// TIA Portal V15.1 export
// export: Created 2020-06-12T07:35:47.8505859Z, ExportSetting None, DisplayName Totally Integrated Automation Portal, DisplayVersion V15.1, DisplayName TIA Portal Openness, DisplayVersion V15.1, DisplayName STEP 7 Professional, DisplayVersion V15.1, DisplayName STEP 7 Safety, DisplayVersion V15.1, DisplayName WinCC Advanced, DisplayVersion V15.1
FUNCTION "DED_Line" : Void   // FC551, FBD
TITLE = Dedusting Pressure control
{ S7_Optimized_Access := 'FALSE' }
// stored: AutoNumber false, SetENOAutomatically False
   VAR_TEMP
      _csf : Bool;
      _hi : Bool;
      _bet : Bool;
      _lo : Bool;
      _cv01_init : Real;
      tVentDemand : Bool;
      _lockw : Word;
      tOpen : Bool;
      tUseIndirect : Bool;
      tLimPressure : Real;
      tCV01set : Real;
      tVarR1 : Real;
      tEnableIndirect : Bool;
      tHoodPressSet : Real;
      tContLock : Bool;
      tContAckn : Bool;
      tContIsOn : Bool;
      tContIsLocked : Bool;
      tContHasFault : Bool;
      tPressAboveSet : Real;
      tDPhigh : Real;
      tCV01set2 : Real;
   END_VAR
   VAR_TEMP   // added for the SCL form of the ladder/FBD networks
      _w1 : Bool;
   END_VAR
BEGIN

REGION Network 1: COMMON SYSTEM FAULT
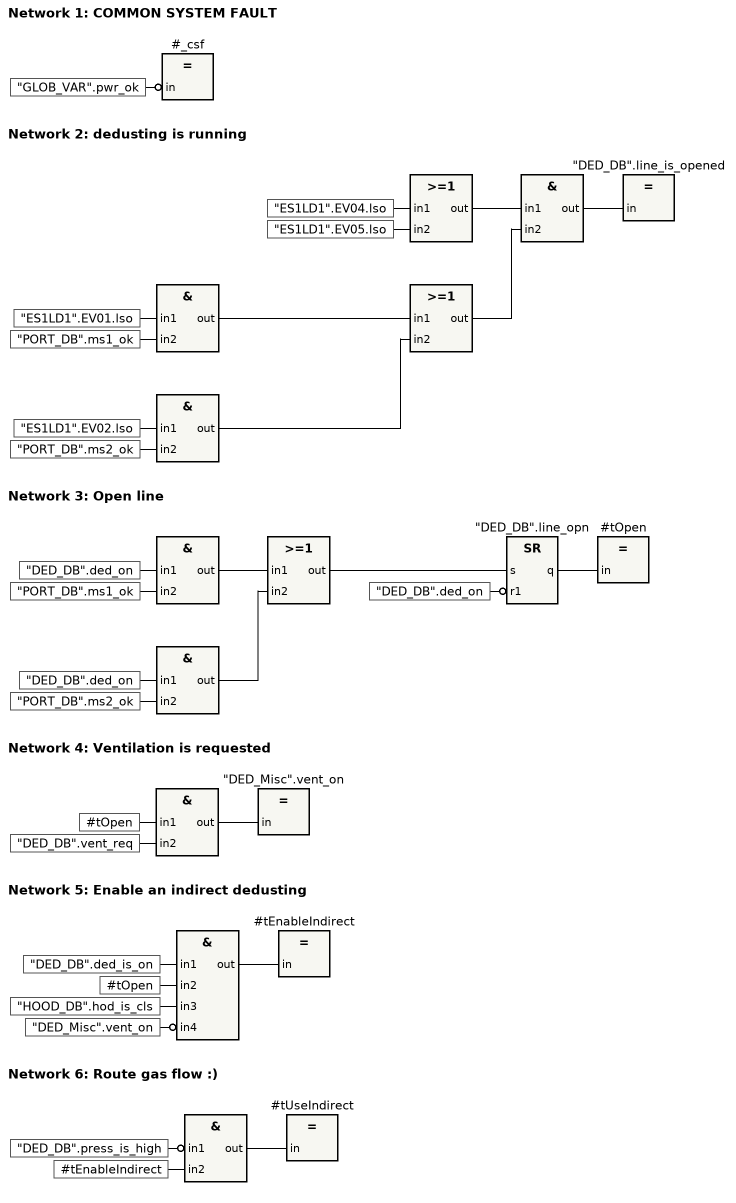
   #_csf := NOT "GLOB_VAR".pwr_ok;
END_REGION

REGION Network 2: dedusting is running
   "DED_DB".line_is_opened := ("ES1LD1".EV04.lso OR "ES1LD1".EV05.lso) AND (("ES1LD1".EV01.lso AND "PORT_DB".ms1_ok) OR ("ES1LD1".EV02.lso AND "PORT_DB".ms2_ok));
END_REGION

REGION Network 3: Open line
   IF ("DED_DB".ded_on AND "PORT_DB".ms1_ok) OR ("DED_DB".ded_on AND "PORT_DB".ms2_ok) THEN
       "DED_DB".line_opn := TRUE;   // SR flip-flop
   END_IF;
   IF NOT "DED_DB".ded_on THEN "DED_DB".line_opn := FALSE; END_IF;
   #tOpen := "DED_DB".line_opn;
END_REGION

REGION Network 4: Ventilation is requested
   "DED_Misc".vent_on := #tOpen AND "DED_DB".vent_req;
END_REGION

REGION Network 5: Enable an indirect dedusting
   #tEnableIndirect := "DED_DB".ded_is_on AND #tOpen AND "HOOD_DB".hod_is_cls AND NOT "DED_Misc".vent_on;
END_REGION

REGION Network 6: Route gas flow :)
   #tUseIndirect := NOT "DED_DB".press_is_high AND #tEnableIndirect;
END_REGION

REGION Network 7: Pressure Tresholds calculation
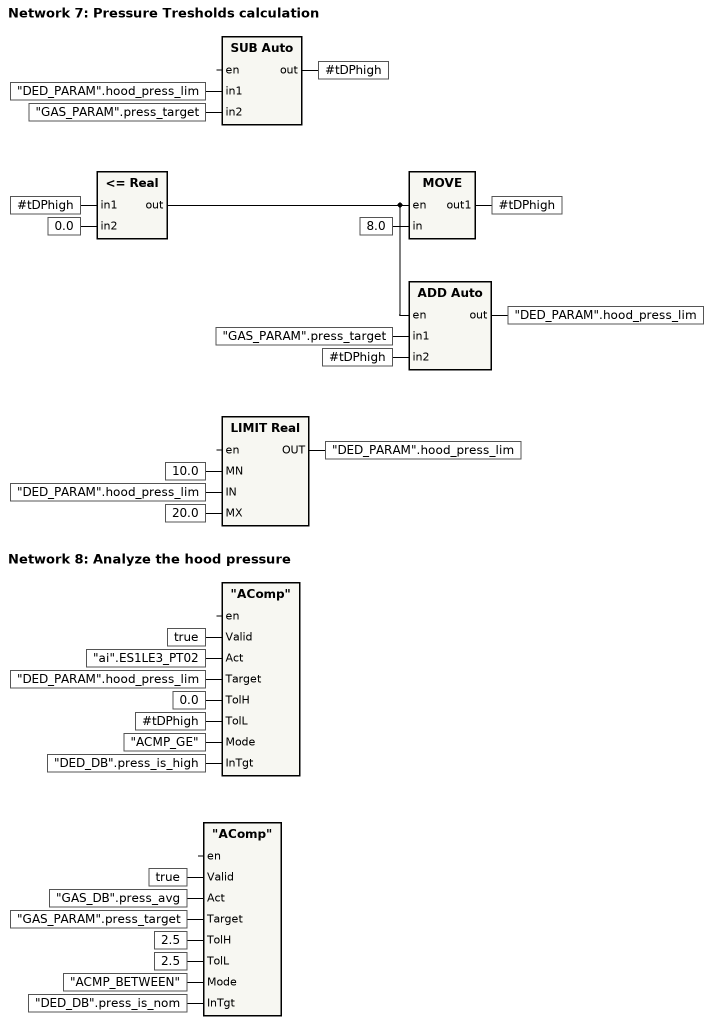
   #tDPhigh := "DED_PARAM".hood_press_lim - "GAS_PARAM".press_target;
   #_w1 := #tDPhigh <= 0.0;
   IF #_w1 THEN
       #tDPhigh := 8.0;
       "DED_PARAM".hood_press_lim := "GAS_PARAM".press_target + #tDPhigh;
   END_IF;
   "DED_PARAM".hood_press_lim := LIMIT(MN := 10.0, IN := "DED_PARAM".hood_press_lim, MX := 20.0);
END_REGION

REGION Network 8: Analyze the hood pressure
   "AComp"(Valid := true,
           Act := "ai".ES1LE3_PT02,
           Target := "DED_PARAM".hood_press_lim,
           TolH := 0.0,
           TolL := #tDPhigh,
           Mode := "ACMP_GE",
           InTgt := "DED_DB".press_is_high);
   "AComp"(Valid := true,
           Act := "GAS_DB".press_avg,
           Target := "GAS_PARAM".press_target,
           TolH := 2.5,
           TolL := 2.5,
           Mode := "ACMP_BETWEEN",
           InTgt := "DED_DB".press_is_nom);
END_REGION

REGION Network 9: Detect the pressure
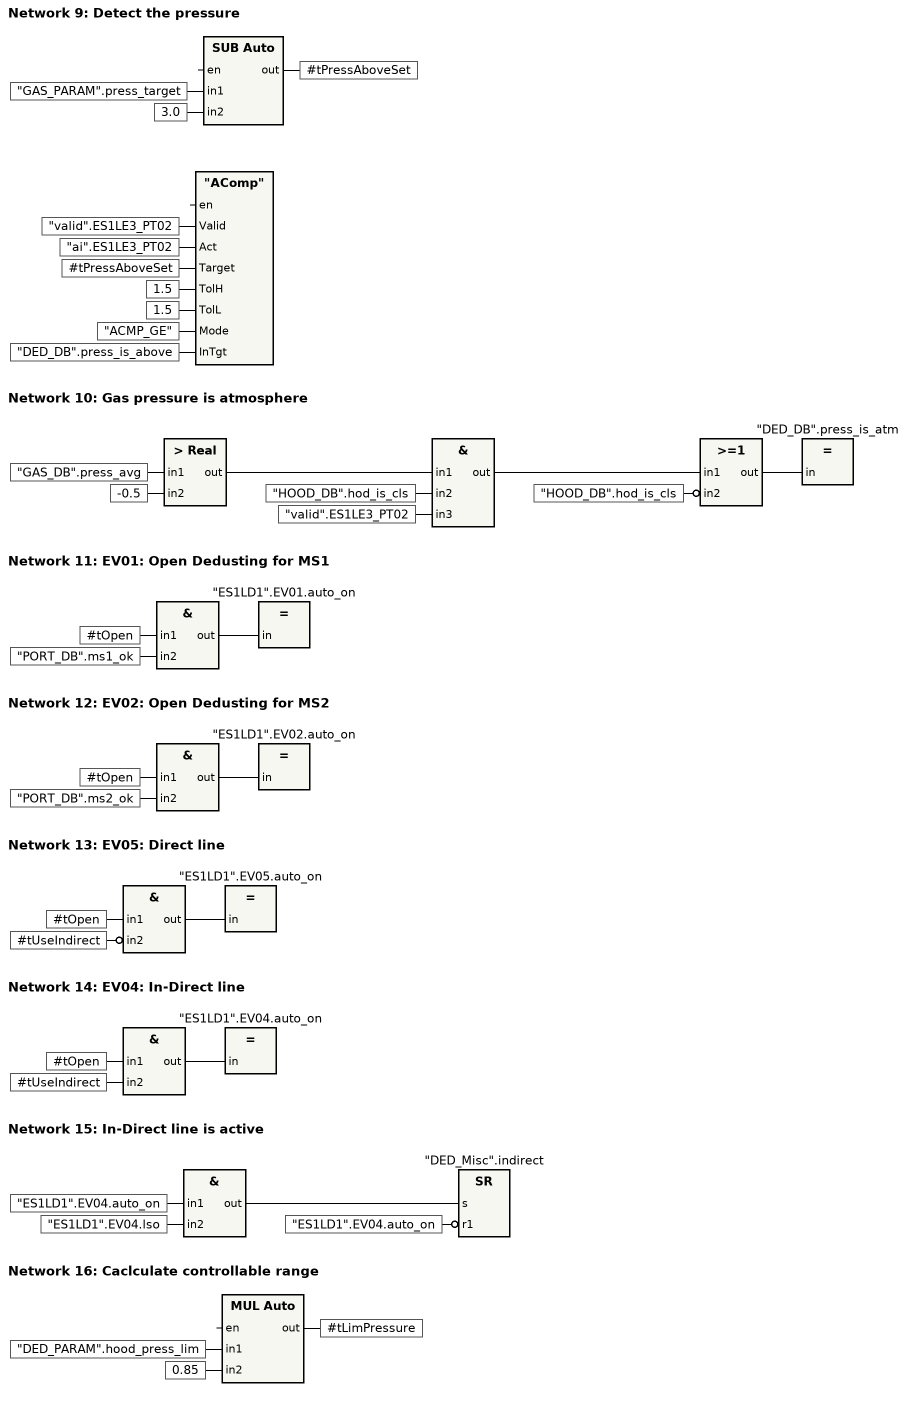
   #tPressAboveSet := "GAS_PARAM".press_target - 3.0;
   "AComp"(Valid := "valid".ES1LE3_PT02,
           Act := "ai".ES1LE3_PT02,
           Target := #tPressAboveSet,
           TolH := 1.5,
           TolL := 1.5,
           Mode := "ACMP_GE",
           InTgt := "DED_DB".press_is_above);
END_REGION

REGION Network 10: Gas pressure is atmosphere
   "DED_DB".press_is_atm := (("GAS_DB".press_avg > (-0.5)) AND "HOOD_DB".hod_is_cls AND "valid".ES1LE3_PT02) OR NOT "HOOD_DB".hod_is_cls;
END_REGION

REGION Network 11: EV01: Open Dedusting for MS1
   "ES1LD1".EV01.auto_on := #tOpen AND "PORT_DB".ms1_ok;
END_REGION

REGION Network 12: EV02: Open Dedusting for MS2
   "ES1LD1".EV02.auto_on := #tOpen AND "PORT_DB".ms2_ok;
END_REGION

REGION Network 13: EV05: Direct line
   "ES1LD1".EV05.auto_on := #tOpen AND NOT #tUseIndirect;
END_REGION

REGION Network 14: EV04: In-Direct line
   "ES1LD1".EV04.auto_on := #tOpen AND #tUseIndirect;
END_REGION

REGION Network 15: In-Direct line is active
   IF "ES1LD1".EV04.auto_on AND "ES1LD1".EV04.lso THEN
       "DED_Misc".indirect := TRUE;   // SR flip-flop
   END_IF;
   IF NOT "ES1LD1".EV04.auto_on THEN "DED_Misc".indirect := FALSE; END_IF;
END_REGION

REGION Network 16: Caclculate controllable range
   #tLimPressure := "DED_PARAM".hood_press_lim * 0.85;
END_REGION

REGION Network 17: Set a pressure with gas blowing
   // I use this to reduce understaing of program :)
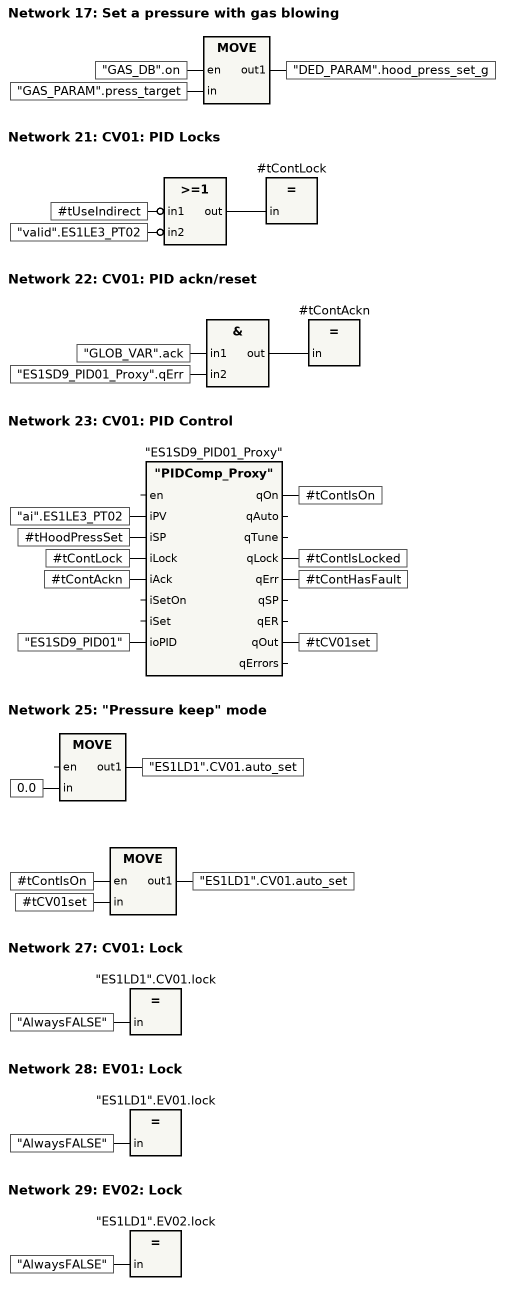
   IF "GAS_DB".on THEN "DED_PARAM".hood_press_set_g := "GAS_PARAM".press_target; END_IF;
END_REGION

REGION Network 18 (SCL): Check and fix the setpoints
   // pressure with gas feeding setpoint 
   "DED_PARAM".hood_press_set_g := ABS("DED_PARAM".hood_press_set_g);
   IF "DED_PARAM".hood_press_set_g < 0.0 THEN
       "DED_PARAM".hood_press_set_g := 0.0;
   ELSIF "DED_PARAM".hood_press_set_g > "DED_PARAM".hood_press_lim THEN
       "DED_PARAM".hood_press_set_g := #tLimPressure;
   END_IF;
   // pressure without gas feeding setpoint 
   "DED_PARAM".hood_press_set_n := ABS("DED_PARAM".hood_press_set_n);
   IF "DED_PARAM".hood_press_set_n < 0.0 THEN
       "DED_PARAM".hood_press_set_n := 0.0;
   ELSIF "DED_PARAM".hood_press_set_n > "DED_PARAM".hood_press_lim THEN
       "DED_PARAM".hood_press_set_n := #tLimPressure;
   END_IF;
END_REGION

REGION Network 19 (SCL): Select the setpoint depends of gas system state
   IF NOT "DED_Misc".vent_on THEN
       #tHoodPressSet := "DED_PARAM".hood_press_set_g;
       IF "Gas_Misc".press_mode THEN
           ;
       END_IF;
       "DED_DB".inlet_press_set := 15.0 - #tHoodPressSet;
   ELSE
       #tHoodPressSet := "DED_PARAM".hood_press_set_n;
       "DED_DB".inlet_press_set := "DED_PARAM".inlet_press_set;
   END_IF;
END_REGION

REGION Network 20: ------
END_REGION

REGION Network 21: CV01: PID Locks
   #tContLock := NOT #tUseIndirect OR NOT "valid".ES1LE3_PT02;
END_REGION

REGION Network 22: CV01: PID ackn/reset
   #tContAckn := "GLOB_VAR".ack AND "ES1SD9_PID01_Proxy".qErr;
END_REGION

REGION Network 23: CV01: PID Control
   // 'ES1SD9PID01 - Dedusting pressure control'
   "ES1SD9_PID01_Proxy"(iPV := "ai".ES1LE3_PT02,   // "PIDComp_Proxy"
                        iSP := #tHoodPressSet,
                        iLock := #tContLock,
                        iAck := #tContAckn,
                        ioPID := "ES1SD9_PID01",
                        qOn => #tContIsOn,
                        qLock => #tContIsLocked,
                        qErr => #tContHasFault,
                        qOut => #tCV01set);
END_REGION

REGION Network 24 (SCL): "Pressure keep" mode (1)
   #tCV01set2 := 50.0 - 8.0 * (#tPressAboveSet - "ai".ES1LE3_PT02);
   IF #tCV01set2 < 0 THEN
       #tCV01set2 := 0.0;
   END_IF;
END_REGION

REGION Network 25: "Pressure keep" mode
   "ES1LD1".CV01.auto_set := 0.0;
   IF #tContIsOn THEN "ES1LD1".CV01.auto_set := #tCV01set; END_IF;
END_REGION

REGION Network 26 (SCL): LD1.CV01 output
   // rlg 27/07/2019 Disable, pressure control was not stable
   //#tVarR1 := #tCV01set / "ES1SC9_PID01".Config.OutputUpperLimit;
   //"ES1LD1".CV01.auto_set := 55.0 + 50.0 * #tVarR1;
   //"ES1LD1".CV01.auto_set := LIMIT_REAL(IN := "ES1LD1".CV01.auto_set
     //                                   , MN := 0.0
       //                                 , MX := 100.0);
END_REGION

REGION Network 27: CV01: Lock
   "ES1LD1".CV01.lock := "AlwaysFALSE";
END_REGION

REGION Network 28: EV01: Lock
   "ES1LD1".EV01.lock := "AlwaysFALSE";
END_REGION

REGION Network 29: EV02: Lock
   "ES1LD1".EV02.lock := "AlwaysFALSE";
END_REGION

REGION Network 30: EV03: Lock
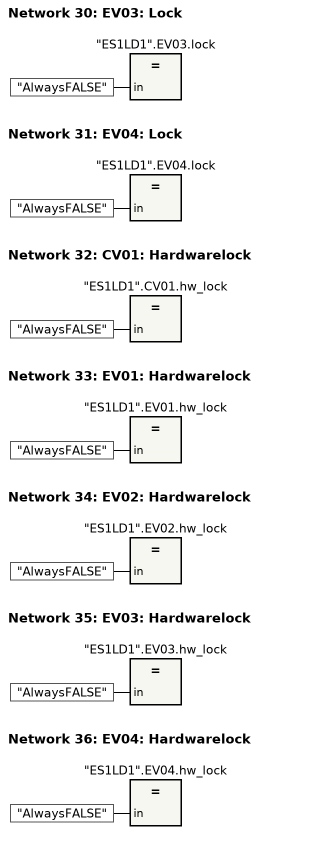
   "ES1LD1".EV03.lock := "AlwaysFALSE";
END_REGION

REGION Network 31: EV04: Lock
   "ES1LD1".EV04.lock := "AlwaysFALSE";
END_REGION

REGION Network 32: CV01: Hardwarelock
   "ES1LD1".CV01.hw_lock := "AlwaysFALSE";
END_REGION

REGION Network 33: EV01: Hardwarelock
   "ES1LD1".EV01.hw_lock := "AlwaysFALSE";
END_REGION

REGION Network 34: EV02: Hardwarelock
   "ES1LD1".EV02.hw_lock := "AlwaysFALSE";
END_REGION

REGION Network 35: EV03: Hardwarelock
   "ES1LD1".EV03.hw_lock := "AlwaysFALSE";
END_REGION

REGION Network 36: EV04: Hardwarelock
   "ES1LD1".EV04.hw_lock := "AlwaysFALSE";
END_REGION
END_FUNCTION
